FUNCTION_BLOCK BLOCK_VVAT_650_ETHERCAT

(* Gestion d'une vanne 3 positions VAT interface ethercat*)

(****************historique des versions*****************************)

(* Version 1-0 - AB - VERSION INITIALE AC2000 - aff 9015 *)
(* Version 2-0 - GV - 06-2015 - affaire 9070 - Adaptation pour journal des évènements externe*)

(*
Configuration vanne : Startup CoE :
Param 0x20F5 _ valeur 0x02 ==> sensor 1 unit à mbar

Configuration vanne via le logiciel VAT CPA , dans terminal :
envoi de la commande 		a:74031 
Cette commande sert à mettre la réception de la pression jauge sur external digital output sensor 1

envoi de la commande			s:2309000000
Cette commande sert à mettre le signal de reception jauge sur un DINT, range par défaut ==> sans doute inutile de la mettre	

Signal de la jauge process envoyée au bloc par entrée I_Pressure (REAL)
Information pression envoyée à la vanne par OUT_Pression_Ethercat (DINT, avec max range de 1 000 000)

*)


(*************************************************************************)


VAR_INPUT
(*paramètre standard*)
	RESET:   					BOOL; 											(*Condition RAZ actionneur*)
	MANUAL:  					BOOL; 	(* ~ (OPC : 1 : available for OPC-clients) *)		(*Mode manuel*)

(*entrée externe*)
	IN_OFF:						BOOL; 	(* ~ (OPC : 1 : available for OPC-clients) *)		(*E.TOR vanne fermée*)
	IN_ON:						BOOL; 	(* ~ (OPC : 1 : available for OPC-clients) *)		(*E.TOR vanne ouverte*)

	IN_POSITION		AT%I*:		DINT;	(*Retour de position de la jauge, de 0 à 100 000 points*)
	I_PRESSION:					REAL;	(*Mesure de pression externe*)

(*Paramètres*)
	PRM_Mode:					BOOL; 	(* ~ (OPC : 1 : available for OPC-clients) *)		(*Mode FALSE = Position / TRUE = Pression*)
	PRM_Pression:				REAL; 	(* ~ (OPC : 1 : available for OPC-clients) *)		(*Consigne de pression - en unité cohérente avec la mesure*)
	PRM_Position:				REAL;	(* ~ (OPC : 1 : available for OPC-clients) *)		(*Consigne de position de la vanne en %*)
	PRM_W_Pr_HI:				REAL;	(* ~ (OPC : 1 : available for OPC-clients) *)		(*Tolérance haute de stabilisation de pression pour obtention de l'état stab pression ok*)
	PRM_W_Pr_LO:				REAL;	(* ~ (OPC : 1 : available for OPC-clients) *)		(*Tolérance basse de dtabilisation de pression pour obtention de l'état stab pression ok*)
	PRM_Tim_W_Pr:				TIME;	(* ~ (OPC : 1 : available for OPC-clients) *)		(*Temps de validation de stabilisation de la pression*)

(*défaut du bloc*)
	DEF_On:  					PRCDEF; 										(*00 - Défaut d'ouverture de la vanne*)
	DEF_Off:   					PRCDEF; 										(*01 - Défaut de fermeture de la vanne*)
	DEF_On_Imposs:				PRCDEF;										(*03 - Défaut d'ouverture ou de mise en laminage non autorisée en mode automatique*)
	DEF_Off_Imposs:				PRCDEF;										(*04 - Défaut de fermeture non autorisée en mode automatique*)
	DEF_Off_auto:				PRCDEF;										(*05 - Défaut de fermeture automatique de la vanne*)
	DEF_Position:				PRCDEF;										(*06 - Défaut d'obtention de la position*)
	DEF_Pression:				PRCDEF;										(*07 - Défaut d'obtention de la pression*)
	DEF_Surv_Pression:			PRCDEF;										(*08 - Défaut de surveillance de la pression - perte du critère de stabilisation*)
	ALA_Surv_Pression:			PRCDEF;										(*09 - Alarme de surveillance de la rpession - perte du critère de stabilisation*)

(*parametre de pilotage en entrée*)
	CO_On:   					BOOL; 											(*Ordre mode automatique ouverture*)
	CO_Lam:						BOOL;											(*Ordre mode automatique laminage*)
	EN_On_INT:   				BOOL;											(*Condition d'autorisation d'ouverture ou de laminage donnée par le bloc qui instancie le bloc actuator*)
	EN_Off_INT:  				BOOL; 											(*Condition d'autorisation de fermeture donnée par le bloc qui instacie le bloc actuator*)
	EN_On_EXT:					BOOL:=TRUE;									(*condition d'autorisation d'ouverture ou de laminage externe*)
	EN_Off_EXT:					BOOL:=TRUE;									(*condition d'autorisation de fermeture externe*)
END_VAR

VAR_INPUT PERSISTENT
(*parametre de configuration constructeur*)
(*les parametres suivants dépendent de la configuration de la machine*)
	CONF_Tim_Valid_On:  		TIME:=T#100MS; 			(*Temps validation de la position ouverte *)
	CONF_Tim_Valid_Off:   		TIME:=T#100ms; 			(*Temps validation de la position fermée *)
	CONF_EN_On:					USINT:=0;				(*définit la réaction du système en cas de perte des conditions d'autorisation d'activation EN_On*)
														(* 0 = désactivation automatique  en cas de perte des conditions d'autorisation d'activation uniquement en manuel*)
														(* 1 = désactivation automatique en cas de perte des conditions d'autorisation d'activation en auto et en manuel*)
														(* 2 = Pas de déscativation automatique*)
	CONF_Pr_Max_SP:			REAL;					(* Consigne max. de pression en pleine echelle 10V - correspond à la pleine échelle du capteur connecté au coffret*)
	CONF_WPos:				REAL;					(*Tolérance de positionnement pour obtention de l'état STATE_POS_ok*)
	CONF_Tim_WPos:			TIME;					(*Temps de validation de l'état STATE_POS_Ok*)
	PRM_Max_Tim_W:			TIME;	(* ~ (OPC : 1 : available for OPC-clients) *)		(*Temps Max d'obtention de l'état stabilisation pression ok*)
	PRM_Tim_Def_Pr:			TIME;	(* ~ (OPC : 1 : available for OPC-clients) *)		(*Temps d'enveloppe du défaut de surveillance de la pression*)
	PRM_Tim_Ala_Pr:			TIME;	(* ~ (OPC : 1 : available for OPC-clients) *)		(*Temps d'enveloppe de l'alarme de surveillance de la pression*)

	(*Entité*)
	IsComponent:	BOOL;			(*entité : composant*)
	IdXML:			STRING;			(*nom entité : identifiant pour recherche dans dico*)
	TagXML:			UINT;			(*nom entité : identifiant pour recherche dans dico*)
	IdParent:		STRING;			(*MNEMO de l'appelant*)
	MNEMO:			STRING;			(*MNEMO de l'entité*)
END_VAR

VAR_OUTPUT
	OUT_Pressure				AT%Q*:	DINT;	(*envoi de la pression reçue par jauge sur trame ethercat, codée sur 1 000 000 point pour pleine échelle*)
	OUT_Control_Mode			AT%Q*:	USINT;	(*control mode : 2-position, 3-close, 4-open, 5-pression*)
	OUT_Pressure_Setpoint		AT%Q*:	DINT;	(*consigne puissance, codé sur 1 000 000 points pour pleine echelle*)
	OUT_Position_Setpoint		AT%Q*:	DINT;	(*consigne position , codé sur 100 000 point pour 100%*)

	STATE_On:	   				BOOL; 	(* ~ (OPC : 1 : available for OPC-clients) *)		(*Indicateur ouverture ok*)
	STATE_Off:  				BOOL; 	(* ~ (OPC : 1 : available for OPC-clients) *)		(*Indicateur fermeture ok*)
	STATE_Nok:					BOOL;	(* ~ (OPC : 1 : available for OPC-clients) *)		(*Indicateur défaut sur la vanne*)
	STATE_Lam:					BOOL;	(* ~ (OPC : 1 : available for OPC-clients) *)		(*Indicateur mise en laminage ok *)
	STATE_Pos_Ok:				BOOL;	(* ~ (OPC : 1 : available for OPC-clients) *)		(*Indicateur de positionnement de la vanne ok *)
	STATE_Press_Ok:				BOOL;	(* ~ (OPC : 1 : available for OPC-clients) *)		(*Indicateur de stabilisation de la pression ok *)
	STATE_Ok:					BOOL;	(* ~ (OPC : 1 : available for OPC-clients) *)		(*Indicateur de stabilisation autour du point de consigne de pression
																				ou de positionnement ok si le controle est en mode position*)
	STATE_Position:				REAL;	(* ~ (OPC : 1 : available for OPC-clients) *)		(*Retour de position de la vanne*)
	STATE_Setpoint:				REAL;	(* ~ (OPC : 1 : available for OPC-clients) *)		(*Valeur de la consigne de pression ou position demandée*)
	STATE_Mode:					BOOL;	(* ~ (OPC : 1 : available for OPC-clients) *)		(*Mode de régulation en cours*)

	AUTOR_On_IHM:				BOOL; 	(* ~ (OPC : 1 : available for OPC-clients) *)		(*etat ouverture autorisée depuis la supervision en mode manuel*)
	AUTOR_Off_IHM:				BOOL; 	(* ~ (OPC : 1 : available for OPC-clients) *)		(*etat fermeture autorisée depuis la supervision en mode manuel*)
	AUTOR_Lam_IHM:				BOOL;	(* ~ (OPC : 1 : available for OPC-clients) *)		(*etat laminage autorisée depuis la supervision en mode manuel*)
	AUTOR_On_PLC:				BOOL;											(*etat ouverture autorisée depuis l'automate*)
	AUTOR_Off_PLC:				BOOL;											(*etat fermeture autorisée depuis l'automate*)
END_VAR


VAR
	(*retours vanne ouvrete fermée selon retour position*)
	VAR_IN_OFF:					BOOL; 	(* retour vanne fermée*)
	VAR_IN_ON:					BOOL; 	(*retour vanne ouverte*)

	TIMER_Valid_On:				TON;
	TIMER_Valid_Off:			TON;
	TIMER_Valid_Pos_ok:			TON;
	TIMER_Valid_Press_ok:		TON;

	M_On:  						BOOL; 	(* ~ (OPC : 1 : available for OPC-clients) *)		(*Ordre mode manuel ouverture de la vanne*)
	M_Off:   					BOOL; 	(* ~ (OPC : 1 : available for OPC-clients) *)		(*Ordre mode manuel fermeture de la vanne*)
	M_Lam:   					BOOL; 	(* ~ (OPC : 1 : available for OPC-clients) *)		(*Ordre mode manuel de mise en position laminage*)
	RCP_M_On:   				BOOL;
	RCP_M_Off:  				BOOL;
	RCP_M_Lam:					BOOL;
	VAR_On:						BOOL;											(*bit intermédiaire de demande d'ouverture de la vanne*)
	VAR_Lam:					BOOL;											(*bit intermédiaire de demande de mise en laminage de la vanne*)
	VAR_Mem_PRM_Pression:		REAL;											(*variable de mémorisation de la consigne de pression*)
	VAR_Prm_Pression_modifie:	BOOL;											(*variable activée à chaque changement de consigne de pression*)
	VAR_Attente_Stab:			BOOL;											(*variable activée aprés chaque demande de changement de consigne lorsque
																				la stabilisation de pression est attendue*)
	VAR_Surv_Pression:			BOOL;											(*variable indiquant que la pression doit être surveillée - stabilisation atteinte*)
END_VAR

VAR_EXTERNAL
	MANUAL_SAFETY_OFF:		BOOL;											(*desactive les sécurités en mode manuel*)
END_VAR

DEF_On.IdXml					:=	'3';
DEF_On.TagXml					:=	2;

DEF_Off.IdXml					:=	'3';
DEF_Off.TagXml					:=	4;

DEF_On_Imposs.IdXml				:=	'3';
DEF_On_Imposs.TagXml			:=	7;

DEF_Off_Imposs.IdXml			:=	'3';
DEF_Off_Imposs.TagXml			:=	9;

DEF_Off_auto.IdXml				:=	'3';
DEF_Off_auto.TagXml				:=	11;

DEF_Position.IdXml				:=	'16';
DEF_Position.TagXml				:=	9;

DEF_Pression.IdXml				:=	'16';
DEF_Pression.TagXml				:=	8;

DEF_Surv_Pression.IdXml			:=	'16';
DEF_Surv_Pression.TagXml		:=	11;

ALA_Surv_Pression.IdXml			:=	'16';
ALA_Surv_Pression.TagXml		:=	10;
ALA_Surv_Pression.Groupe		:=	1;

(*Traitement du signal d'entrée de position codé sur 100 000 points pour 100%*)
STATE_Position	:=	DINT_TO_REAL(IN_POSITION / 1000);
(*Envoi de la pression de la jauge vers la vanne*)
OUT_Pressure	:=	REAL_TO_DINT(I_PRESSION * 1000000 / CONF_Pr_Max_SP);


(*Mémorisation de la consigne et détection de changement de consigne*)
VAR_Prm_Pression_modifie :=  (PRM_Pression <> VAR_Mem_PRM_pression) AND VAR_Lam AND PRM_MODE AND NOT MANUAL AND NOT RESET;;
IF VAR_Lam AND PRM_mode THEN
	VAR_Mem_PRM_Pression	:= PRM_Pression;
ELSE
	VAR_Mem_PRM_Pression := 0.0;
END_IF;
(*positionnement du bit d'attente de la stabilisation de pression aprés modification de la consigne de pression*)
IF VAR_Prm_Pression_modifie AND NOT MANUAL AND NOT RESET  THEN
	VAR_Attente_Stab := TRUE;
END_IF;

(* Réception des ordres en mode manuel*)
RCP_M_On 			:=	M_On;
RCP_M_Off			:=	M_Off;
RCP_M_Lam			:=	M_Lam;

(*Autorisation*)
AUTOR_On_IHM		:= 	MANUAL AND ((EN_On_INT AND EN_On_EXT)
						OR MANUAL_SAFETY_OFF) AND NOT RESET AND NOT VAR_On;
AUTOR_Off_IHM		:= 	MANUAL AND ((EN_Off_INT AND EN_Off_EXT)  OR
						MANUAL_SAFETY_OFF) AND NOT RESET AND  (VAR_On OR VAR_Lam);
AUTOR_Lam_IHM	:=	MANUAL AND ((EN_On_INT AND EN_On_EXT)
						OR MANUAL_SAFETY_OFF) AND NOT RESET AND NOT VAR_Lam;
AUTOR_On_PLC		:=	NOT MANUAL AND (EN_On_INT AND EN_On_EXT)
						AND NOT RESET;
AUTOR_Off_PLC		:= 	NOT MANUAL AND (EN_Off_INT AND EN_Off_EXT)
						AND NOT RESET;
(*defaut ouverture ou laminage impossible en mode automatique*)
DEF_On_Imposs.CONDITION:=	(CO_On OR CO_Lam) AND NOT AUTOR_On_PLC AND NOT MANUAL;
DEF_On_Imposs.DELAY := T#0ms;
DEF_On_Imposs();
(*Defaut fermeture impossible en mode automatique*)
DEF_Off_Imposs.CONDITION:=	NOT CO_On AND NOT CO_Lam AND NOT AUTOR_Off_PLC AND NOT MANUAL
							AND (VAR_Lam OR VAR_On);
DEF_Off_Imposs.DELAY := T#0ms;
DEF_Off_Imposs();
(*defaut de fermeture automatique de la vanne*)
DEF_Off_Auto.CONDITION :=             (NOT EN_On_INT OR NOT EN_On_EXT) AND  (VAR_On OR VAR_Lam)
								 AND ((CONF_En_ON=1) OR ((CONF_EN_On=0) AND MANUAL)) AND NOT RESET;
DEF_Off_auto.DELAY:=T#0ms;
DEF_Off_Auto();

(*gestion des sorties*)
IF 		(RCP_M_On AND AUTOR_On_IHM) OR
		(CO_On AND AUTOR_On_PLC) THEN
				VAR_On		:= 	TRUE;
				VAR_Lam	:= 	FALSE;
ELSIF 	(RCP_M_Lam AND AUTOR_Lam_IHM) OR
	    	(CO_Lam AND AUTOR_On_PLC) THEN
				VAR_On		:=	FALSE;
				VAR_LAm	:=	TRUE;
ELSIF 	RESET  OR DEF_Off_Auto.DEF OR
		(RCP_M_Off AND AUTOR_Off_IHM) OR
	    	((NOT CO_Lam AND NOT CO_On) AND AUTOR_Off_PLC) THEN
				VAR_On		:= 	FALSE;
				VAR_Lam	:=	FALSE;
END_IF;

(*Gestion du control mode*)
(*Ouverture vanne*)
IF VAR_ON THEN
	OUT_Control_Mode := 4;
END_IF;
(*fermeture vanne*)
IF NOT Var_Lam AND NOT Var_on THEN
	OUT_Control_Mode := 3;
END_IF;
(*régulation pression*)
IF Var_Lam AND PRM_MODE THEN
	OUT_Control_Mode := 5;
END_IF;
(*régulation position*)
IF Var_Lam AND NOT Prm_mode THEN
	OUT_Control_Mode := 2;
END_IF;


(*------Gestion de la consigne analogique pression ou position-----*)
(*Envoi de la consigne de pression*)
IF 		PRM_Mode AND VAR_Lam THEN
			OUT_Pressure_Setpoint	:=	REAL_TO_DINT(PRM_Pression * 1000000 / CONF_Pr_Max_SP);
			STATE_Mode	:=	TRUE;
(*Envoi de la consigne de position*)
ELSIF 	NOT PRM_Mode AND VAR_Lam THEN
			OUT_Position_Setpoint	:=	REAL_TO_DINT(PRM_Position * 1000);
			STATE_Mode	:=	FALSE;
(*RaZ des consignes*)
ELSIF NOT VAR_Lam	THEN
			OUT_Position_Setpoint	:=	0;
			OUT_Pressure_Setpoint	:=	0;
END_IF;


(*Retour vanne ouverte fermée selon position*)
VAR_IN_OFF := (State_position = 0) ;
VAR_IN_ON := (State_position = 100) ;



(*indicateur actionneur activé STATE_ON*)
TIMER_Valid_On.IN	:=	VAR_ON AND VAR_IN_On;
TIMER_Valid_On(PT:=CONF_Tim_Valid_On);
STATE_ON			:=	TIMER_Valid_On.Q;
(*indicateur actionneur activé STATE_OFF*)
TIMER_Valid_Off.IN	:=	NOT VAR_Lam AND NOT VAR_On AND VAR_IN_off;
TIMER_Valid_Off(PT:=CONF_Tim_Valid_Off);
STATE_Off			:=	TIMER_Valid_Off.Q;
(*indicateur STATE_NOK*)
STATE_Nok			:=	DEF_ON.DEF OR DEF_Off.DEF OR DEF_Off_auto.DEF OR DEF_On_Imposs.DEF OR
						DEF_Off_Imposs.DEF OR DEF_pression.DEF OR DEF_Position.DEF;

(*temporisation de validation de la stabilisation à la consigne de position*)
TIMER_Valid_Pos_OK.IN		:=	VAR_Lam AND NOT PRM_Mode AND(  (ABS(STATE_Position - PRM_position) <= CONF_WPos) OR (CONF_WPos = 0.0));
TIMER_Valid_Pos_OK.PT		:=	CONF_Tim_WPos;
Timer_Valid_pos_OK();
STATE_Pos_OK				:= 	TIMER_Valid_Pos_OK.Q;


(*temporisation de validation de la stabilisation à la consigne de pression*)
TIMER_Valid_Press_OK.IN		:=	VAR_Lam AND PRM_Mode AND (((I_Pression >= PRM_W_Pr_LO) AND (I_Pression <= PRM_W_Pr_HI))
								OR (PRM_Tim_W_Pr = T#0ms))
								AND NOT VAR_Prm_Pression_modifie ;
TIMER_Valid_Press_OK.PT		:=	PRM_Tim_W_Pr;
TIMER_Valid_Press_OK();
STATE_Press_OK				:=	TIMER_Valid_Press_ok.Q;

(*indicateur actionneur activé STATE_LAM*)
STATE_Lam			:=	(VAR_Lam AND PRM_Mode) OR (VAR_LAM AND NOT PRM_Mode AND STATE_Pos_ok);
STATE_Ok  			:= 	STATE_Pos_Ok OR STATE_Press_Ok;

(*positionnement du bit de validation de la surveillance de la pression
si la stabilisation de pression est obtenue*)
IF (VAR_Lam AND PRM_MODE AND STATE_Press_ok) AND NOT MANUAL AND NOT RESET  THEN
	VAR_Surv_Pression :=	TRUE;
END_IF;
(*RAZ du bit d'attente de la stabilisation de pression lorsque l'état de stabilisation pression a été atteint ou
que le mode régulation de pression n'est plus demandé*)
IF (VAR_Attente_stab AND STATE_Press_ok) OR RESET OR NOT (VAR_Lam AND PRM_Mode)  THEN
	VAR_Attente_Stab := FALSE;
END_IF;

(*RAZ du bit de surveillance de la stabilisation si pas en mode régulation de pression ou si un changement de consigne est apparu*)
IF VAR_Prm_Pression_modifie  OR RESET OR NOT (VAR_Lam AND PRM_Mode)  THEN
	VAR_Surv_Pression := FALSE;
END_IF;

(*défaut d'ouverture*)
DEF_On.Condition		:= 	VAR_On AND NOT STATE_On;
DEF_On();
(*défaut de fermeture*)
DEF_Off.Condition		:= 	NOT VAR_on AND NOT VAR_Lam AND NOT STATE_Off;
DEF_Off();
(*défaut d'obtention de la position*)
DEF_Position.Condition	:= 	VAR_Lam AND NOT PRM_Mode AND NOT STATE_Pos_Ok;
DEF_position();
(*défaut d'obtention de la pression - le défaut n'est plus surveillé lorsque l'état STATE_Press_ok a été atteint  et est
surveillé de nouveau aprés un changement de consigne*)
DEF_Pression.Condition	:= 	VAR_Lam AND PRM_Mode AND NOT STATE_Press_Ok AND VAR_Attente_Stab
							AND NOT MANUAL AND NOT RESET;
DEF_Pression(DELAY		:=	PRM_Max_Tim_W);

(*défaut de surveillance de la pression - l'état STATE_Press_Ok est perdu pendant un temps supérieur à PRM_TIM_SURV_PR *)
DEF_Surv_Pression.CONDITION	:=	VAR_Lam AND PRM_Mode AND NOT State_Press_OK AND VAR_Surv_Pression
								AND NOT MANUAL AND NOT RESET;
DEF_Surv_Pression (DELAY:=PRM_Tim_Def_Pr);


(*défaut de surveillance de la pression - l'état STATE_Press_Ok est perdu pendant un temps supérieur à PRM_ALA_SURV_PR*)
ALA_Surv_Pression.CONDITION 	:=	VAR_Lam AND PRM_Mode AND NOT State_Press_OK AND VAR_Surv_Pression
									AND NOT MANUAL AND NOT RESET;
ALA_Surv_Pression (DELAY:=PRM_Tim_Ala_Pr);

(* Reset des ordres *)
IF M_On AND RCP_M_On THEN
	M_On 	:= FALSE;
END_IF;
IF M_Off AND RCP_M_Off THEN
	M_Off		 := FALSE;
END_IF;
IF M_Lam AND RCP_M_Lam THEN
	M_Lam		 := FALSE;
END_IF;

END_FUNCTION_BLOCK

(* stored: Version 1.1.0.1, ProductVersion 3.1.4024.10
   POU BLOCK_VVAT_650_ETHERCAT: Id {2879890a-0625-4952-b142-20684aacb3d8}, SpecialFunc None *)
